// TIA Portal V20 export
FUNCTION "Service_Tempering" : Void   // FC13, FBD
TITLE = Service
{ S7_Optimized_Access := 'TRUE' }
AUTHOR : Siemens AG
FAMILY : ServiceControl
VERSION : 1.0
// stored: SetENOAutomatically false
   VAR_TEMP
      Temp_TimeMs : DInt;
      Temp_TimeSec : DInt;
      State : "Service_States";
   END_VAR
BEGIN

REGION Network 1: Cm FIC100 feedback
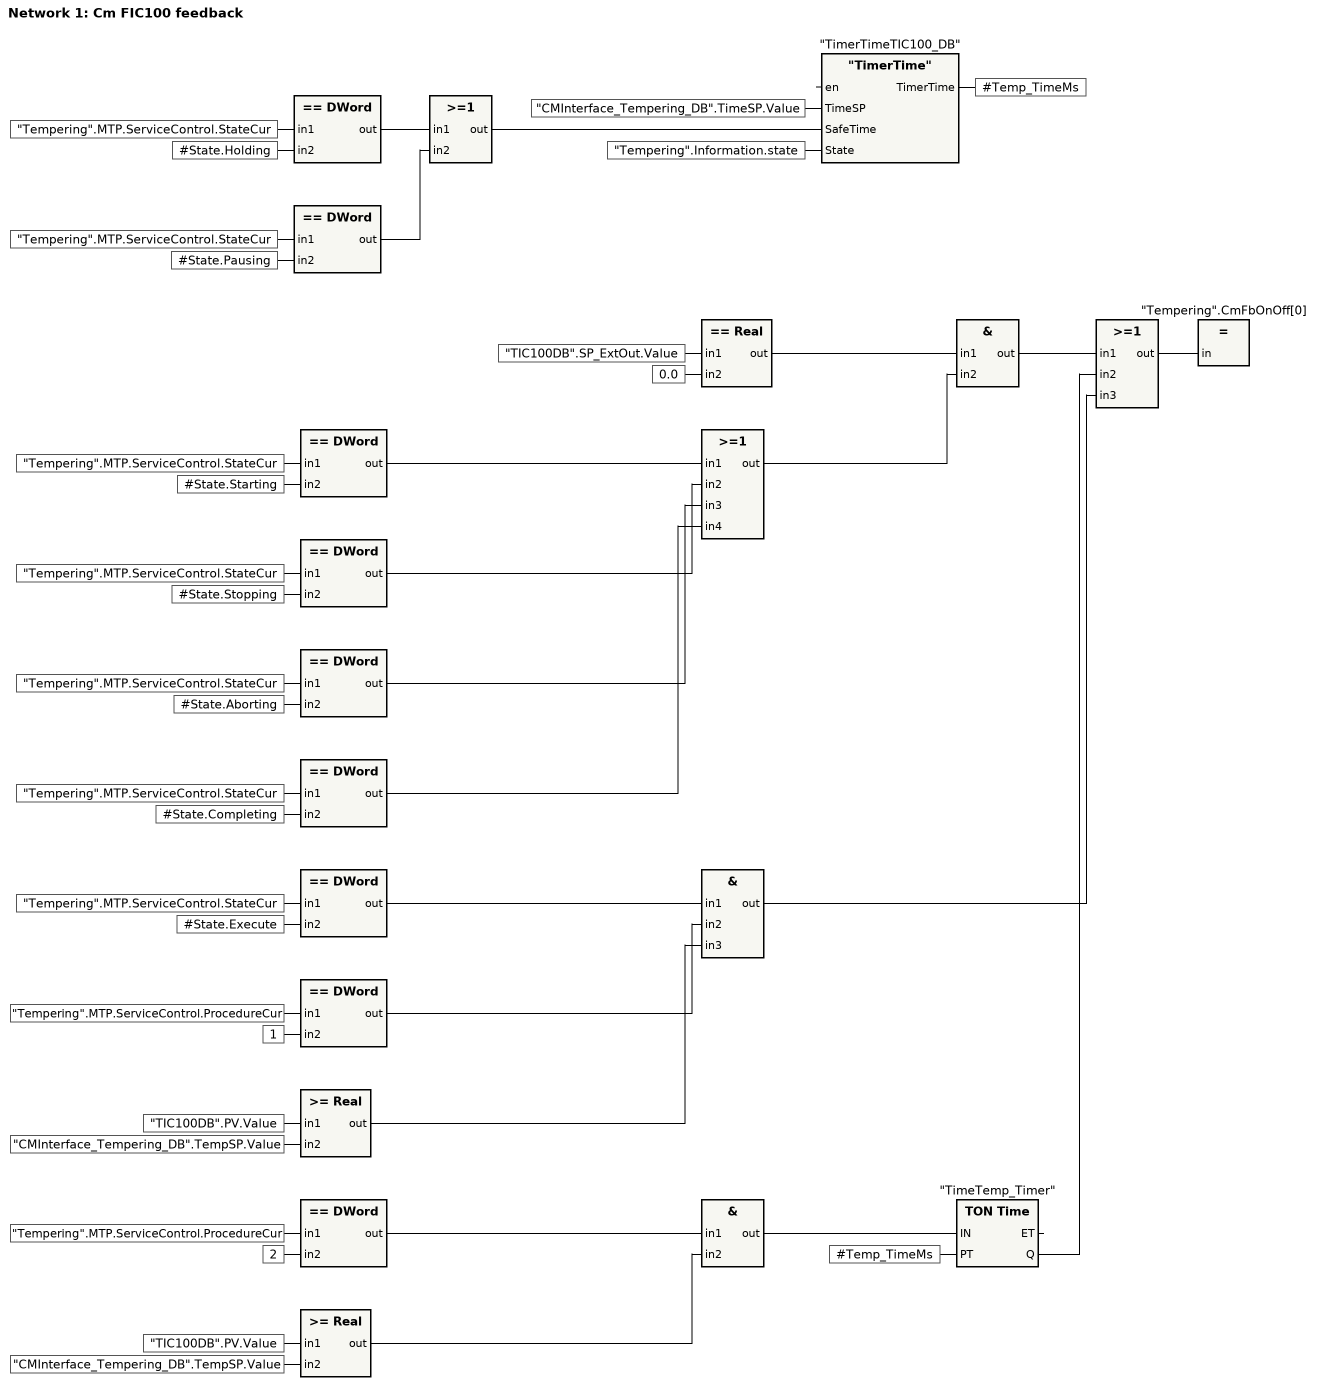
   "TimerTimeTIC100_DB"(TimeSP := "CMInterface_Tempering_DB".TimeSP.Value,   // "TimerTime"
                        SafeTime := ("Tempering".MTP.ServiceControl.StateCur = #State.Holding) OR ("Tempering".MTP.ServiceControl.StateCur = #State.Pausing),
                        State := "Tempering".Information.state,
                        TimerTime => #Temp_TimeMs);
   "TimeTemp_Timer".TON(IN := ("Tempering".MTP.ServiceControl.ProcedureCur = 2) AND ("TIC100DB".PV.Value >= "CMInterface_Tempering_DB".TempSP.Value),
                        PT := #Temp_TimeMs);
   "Tempering".CmFbOnOff[0] := (("TIC100DB".SP_ExtOut.Value = 0.0) AND (("Tempering".MTP.ServiceControl.StateCur = #State.Starting) OR ("Tempering".MTP.ServiceControl.StateCur = #State.Stopping) OR ("Tempering".MTP.ServiceControl.StateCur = #State.Aborting) OR ("Tempering".MTP.ServiceControl.StateCur = #State.Completing))) OR "TimeTemp_Timer".Q OR (("Tempering".MTP.ServiceControl.StateCur = #State.Execute) AND ("Tempering".MTP.ServiceControl.ProcedureCur = 1) AND ("TIC100DB".PV.Value >= "CMInterface_Tempering_DB".TempSP.Value));
END_REGION

REGION Network 2: Set readyToComplete
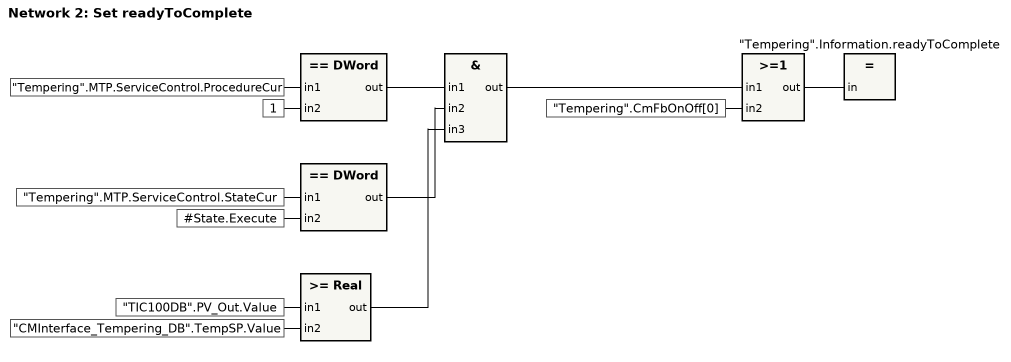
   "Tempering".Information.readyToComplete := (("Tempering".MTP.ServiceControl.ProcedureCur = 1) AND ("Tempering".MTP.ServiceControl.StateCur = #State.Execute) AND ("TIC100DB".PV_Out.Value >= "CMInterface_Tempering_DB".TempSP.Value)) OR "Tempering".CmFbOnOff[0];
END_REGION

REGION Network 3: Service
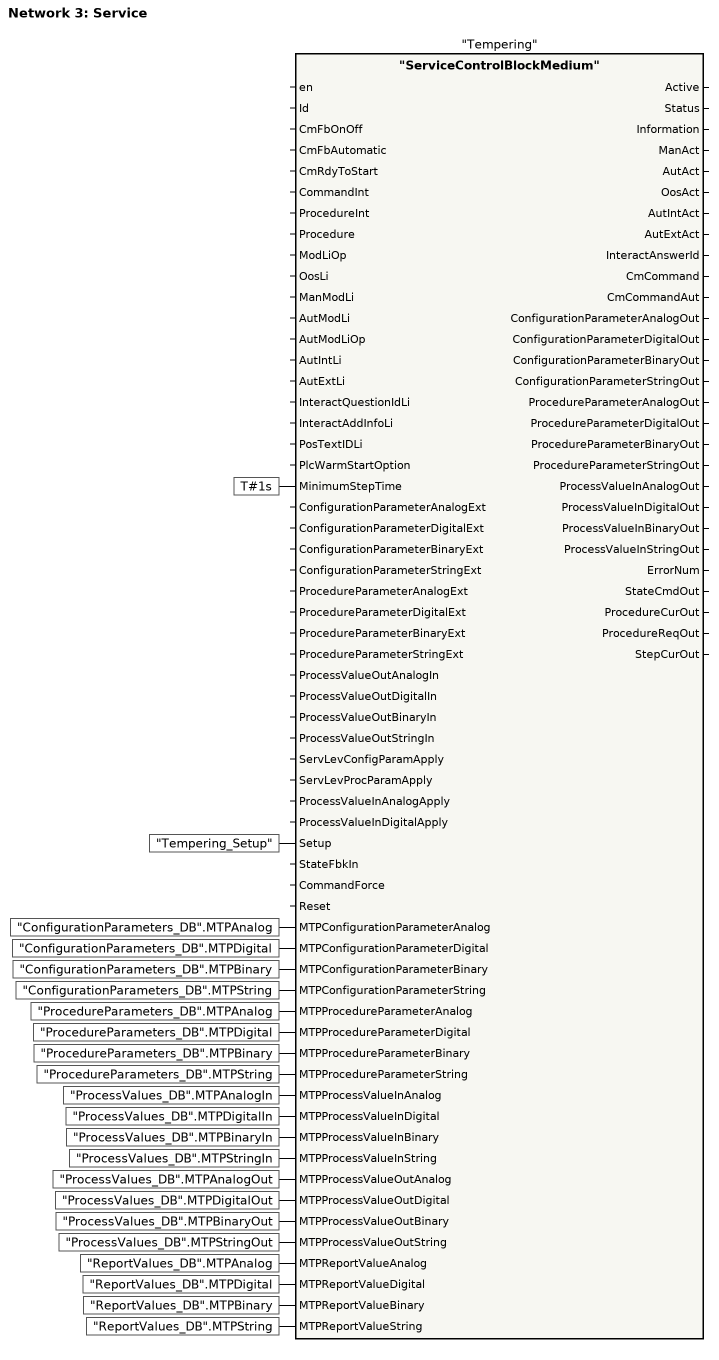
   "Tempering"(MinimumStepTime := T#1s,   // "ServiceControlBlockMedium"
               Setup := "Tempering_Setup",
               MTPConfigurationParameterAnalog := "ConfigurationParameters_DB".MTPAnalog,
               MTPConfigurationParameterDigital := "ConfigurationParameters_DB".MTPDigital,
               MTPConfigurationParameterBinary := "ConfigurationParameters_DB".MTPBinary,
               MTPConfigurationParameterString := "ConfigurationParameters_DB".MTPString,
               MTPProcedureParameterAnalog := "ProcedureParameters_DB".MTPAnalog,
               MTPProcedureParameterDigital := "ProcedureParameters_DB".MTPDigital,
               MTPProcedureParameterBinary := "ProcedureParameters_DB".MTPBinary,
               MTPProcedureParameterString := "ProcedureParameters_DB".MTPString,
               MTPProcessValueInAnalog := "ProcessValues_DB".MTPAnalogIn,
               MTPProcessValueInDigital := "ProcessValues_DB".MTPDigitalIn,
               MTPProcessValueInBinary := "ProcessValues_DB".MTPBinaryIn,
               MTPProcessValueInString := "ProcessValues_DB".MTPStringIn,
               MTPProcessValueOutAnalog := "ProcessValues_DB".MTPAnalogOut,
               MTPProcessValueOutDigital := "ProcessValues_DB".MTPDigitalOut,
               MTPProcessValueOutBinary := "ProcessValues_DB".MTPBinaryOut,
               MTPProcessValueOutString := "ProcessValues_DB".MTPStringOut,
               MTPReportValueAnalog := "ReportValues_DB".MTPAnalog,
               MTPReportValueDigital := "ReportValues_DB".MTPDigital,
               MTPReportValueBinary := "ReportValues_DB".MTPBinary,
               MTPReportValueString := "ReportValues_DB".MTPString);
END_REGION

REGION Network 4: Service HMI
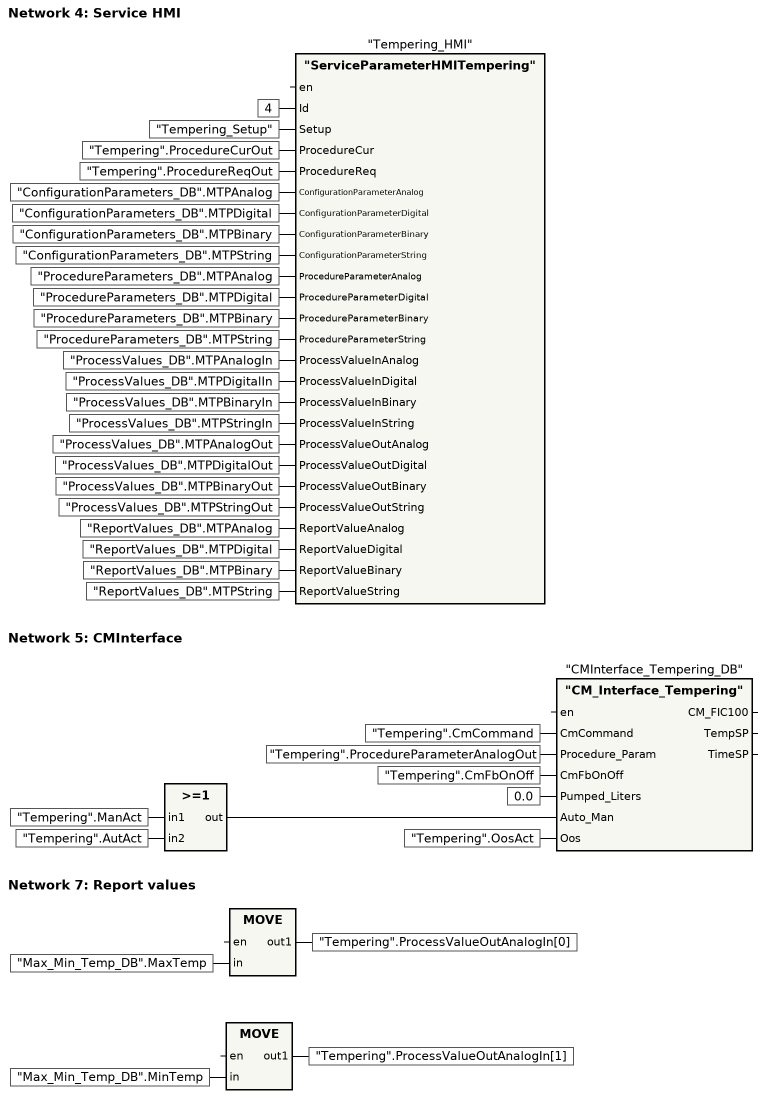
   "Tempering_HMI"(Id := 4,   // "ServiceParameterHMITempering"
                   Setup := "Tempering_Setup",
                   ProcedureCur := "Tempering".ProcedureCurOut,
                   ProcedureReq := "Tempering".ProcedureReqOut,
                   ConfigurationParameterAnalog := "ConfigurationParameters_DB".MTPAnalog,
                   ConfigurationParameterDigital := "ConfigurationParameters_DB".MTPDigital,
                   ConfigurationParameterBinary := "ConfigurationParameters_DB".MTPBinary,
                   ConfigurationParameterString := "ConfigurationParameters_DB".MTPString,
                   ProcedureParameterAnalog := "ProcedureParameters_DB".MTPAnalog,
                   ProcedureParameterDigital := "ProcedureParameters_DB".MTPDigital,
                   ProcedureParameterBinary := "ProcedureParameters_DB".MTPBinary,
                   ProcedureParameterString := "ProcedureParameters_DB".MTPString,
                   ProcessValueInAnalog := "ProcessValues_DB".MTPAnalogIn,
                   ProcessValueInDigital := "ProcessValues_DB".MTPDigitalIn,
                   ProcessValueInBinary := "ProcessValues_DB".MTPBinaryIn,
                   ProcessValueInString := "ProcessValues_DB".MTPStringIn,
                   ProcessValueOutAnalog := "ProcessValues_DB".MTPAnalogOut,
                   ProcessValueOutDigital := "ProcessValues_DB".MTPDigitalOut,
                   ProcessValueOutBinary := "ProcessValues_DB".MTPBinaryOut,
                   ProcessValueOutString := "ProcessValues_DB".MTPStringOut,
                   ReportValueAnalog := "ReportValues_DB".MTPAnalog,
                   ReportValueDigital := "ReportValues_DB".MTPDigital,
                   ReportValueBinary := "ReportValues_DB".MTPBinary,
                   ReportValueString := "ReportValues_DB".MTPString);
END_REGION

REGION Network 5: CMInterface
   "CMInterface_Tempering_DB"(CmCommand := "Tempering".CmCommand,   // "CM_Interface_Tempering"
                           Procedure_Param := "Tempering".ProcedureParameterAnalogOut,
                           CmFbOnOff := "Tempering".CmFbOnOff,
                           Pumped_Liters := 0.0,
                           Auto_Man := "Tempering".ManAct OR "Tempering".AutAct,
                           Oos := "Tempering".OosAct);
END_REGION

REGION Network 6: Block pause and hold state
END_REGION

REGION Network 7: Report values
   "Tempering".ProcessValueOutAnalogIn[0] := "Max_Min_Temp_DB".MaxTemp;
   "Tempering".ProcessValueOutAnalogIn[1] := "Max_Min_Temp_DB".MinTemp;
END_REGION
END_FUNCTION
